FUNCTION_BLOCK PicAlphaConveyor EXTENDS Conveyor
VAR_INPUT
END_VAR
VAR_OUTPUT
END_VAR
VAR
	//Sensors
	m_PresencesensorStart : PresenceSensor;
	m_PresencesensorEnd : PresenceSensor;
	
	m_Switch: Switch;
	m_WPNumberAtPAC : INT := 0;
END_VAR

METHOD METH_IncreaseWPNumberAtPAC : BOOL
VAR_INPUT
END_VAR
m_WPNumberAtPAC := m_WPNumberAtPAC + 1;
END_METHOD

METHOD METH_ReduceWPNumberAtPAC : BOOL
VAR_INPUT
END_VAR
m_WPNumberAtPAC := m_WPNumberAtPAC - 1;
END_METHOD

METHOD METH_ResetWPNumberAtPAC : BOOL
VAR_INPUT
END_VAR
m_WPNumberAtPAC := 0;
END_METHOD

METHOD METH_Switch_Extend : BOOL
VAR_INPUT
END_VAR
m_Switch.METH_Extend();
END_METHOD

METHOD METH_Switch_Retract : BOOL
VAR_INPUT
END_VAR
m_Switch.METH_Retract();
END_METHOD

PROPERTY WPAtEnd : BOOL
GET
WPAtEnd := m_presenceSensorEnd.Value;
END_GET
END_PROPERTY

PROPERTY WPAtStart : BOOL
GET
WPAtStart := m_presenceSensorStart.Value;
END_GET
END_PROPERTY

END_FUNCTION_BLOCK

(* stored: Version 1.1.0.1
   POU PicAlphaConveyor: Id {5ac34ee8-f198-4d86-a5c9-b6b9c7c1e574}, SpecialFunc None
   Folder Methods: Id {29d6a227-c1a9-4e33-8315-e41c44544cda}
   Folder Properties: Id {62eeeee4-90fc-4e30-8dea-689a4b649005}
   Method METH_IncreaseWPNumberAtPAC: Id {0027a79b-0c46-4460-9992-915778e874de}
   Method METH_ReduceWPNumberAtPAC: Id {b6c7e54c-df43-410c-899e-9bcb293db6f3}
   Method METH_ResetWPNumberAtPAC: Id {aedf9399-9da5-4c00-b66a-a27637387329}
   Method METH_Switch_Extend: Id {4728c127-f187-4b87-9218-30de937ef807}
   Method METH_Switch_Retract: Id {de29a4f8-c416-4f7d-a2e8-37aaa8db14ac}
   Property WPAtEnd: Id {8c34190d-dd00-46af-92f3-f9050f60da9f}
   Get Get: Id {1041796b-6338-4c98-b098-b4d410d274b4}
   Property WPAtStart: Id {add39517-8066-4e12-9810-e7bb2e33c739}
   Get Get: Id {72aa0973-9c25-4539-be4f-e2b902c1403e} *)
